// TIA Portal V17 export
// export: Created 2022-07-20T07:01:32.5794371Z, ExportSetting WithDefaults, DisplayName Totally Integrated Automation Portal, DisplayVersion V17, DisplayName TIA Portal Openness, DisplayVersion V17, DisplayName TIA Portal Version Control Interface, DisplayVersion V17, DisplayName SINAMICS Startdrive Advanced, DisplayVersion V17, DisplayName SINAMICS Startdrive G130, G150, S120, S150, SINAMICS MV, S210, DisplayVersion V17, DisplayName SINAMICS Startdrive G110M, G120, G120C, G120D, G120P, G115D, DisplayVersion V17, DisplayName STEP 7 Professional, DisplayVersion V17, DisplayName STEP 7 Safety, DisplayVersion V17, DisplayName WinCC Advanced, DisplayVersion V17
FUNCTION_BLOCK "FB10344_WebGuideProfinet"   // FB10344, LAD
TITLE = FB10342_WebGuide
{ S7_Optimized_Access := 'TRUE' }
VERSION : 0.1
// stored: AutoNumber false, IsIECCheckEnabled false, IsRetainMemResEnabled false, MemoryReserve 100, SetENOAutomatically false, UDAEnableTagReadback false
   VAR_INPUT
      RequestAcknowledge : Bool;
      Parameters : "stWebGuidePNParameters";
      CommInWebGuide_0 : Int;
      CommInWebGuide_1 : Int;
      CommInWebGuide_2 : Int;
      CommInWebGuide_3 : Int;
      CommInWebGuide_4 : Int;
      CommInWebGuide_5 : Int;
      CommInWebGuide_6 : Int;
      CommInWebGuide_7 : Int;
      CommInWebGuide_8 : Int;
      CommInWebGuide_9 : Int;
      CommInWebGuide_10 : Int;
      CommInWebGuide_11 : Int;
      CommInWebGuide_12 : Int;
      CommInWebGuide_13 : Int;
      CommInWebGuide_14 : Int;
      CommInWebGuide_15 : Int;
      CommInWebGuide_16 : Int;
      CommInWebGuide_17 : Int;
      CommInWebGuide_18 : Int;
      CommInWebGuide_19 : Int;
      CommInWebGuide_20 : Int;
      CommInWebGuide_21 : Int;
      CommInWebGuide_22 : Int;
      CommInWebGuide_23 : Int;
      CommInWebGuide_24 : Int;
      CommInWebGuide_25 : Int;
      CommInWebGuide_26 : Int;
      CommInWebGuide_27 : Int;
      CommInWebGuide_28 : Int;
   END_VAR
   VAR_OUTPUT
      CommOutWebGuide_0 : Int;
      CommOutWebGuide_1 : Int;
      CommOutWebGuide_2 : Int;
      CommOutWebGuide_3 : Int;
      CommOutWebGuide_4 : Int;
      CommOutWebGuide_5 : Int;
      CommOutWebGuide_6 : Int;
      CommOutWebGuide_7 : Int;
      CommOutWebGuide_8 : Int;
      CommOutWebGuide_9 : Int;
      CommOutWebGuide_10 : Int;
      CommOutWebGuide_11 : Int;
      CommOutWebGuide_12 : Int;
      CommOutWebGuide_13 : Int;
      CommOutWebGuide_14 : Int;
      CommOutWebGuide_15 : Int;
      CommOutWebGuide_16 : Int;
      CommOutWebGuide_17 : Int;
      CommOutWebGuide_18 : Int;
      CommOutWebGuide_19 : Int;
      CommOutWebGuide_20 : Int;
      CommOutWebGuide_21 : Int;
      CommOutWebGuide_22 : Int;
      CommOutWebGuide_23 : Int;
      CommOutWebGuide_24 : Int;
      CommOutWebGuide_25 : Int;
      CommOutWebGuide_26 : Int;
      CommOutWebGuide_27 : Int;
      CommOutWebGuide_28 : Int;
   END_VAR
   VAR_IN_OUT
      Requests : "stWebGuidePNRequests";
      States : "stWebGuidePNStates";
   END_VAR
   VAR
      RequestInternTrigger : Bool;
      R_Trig_Trigger : R_TRIG;
   END_VAR
BEGIN

REGION Network 1 (SCL): First Scan
   IF "FirstScan" THEN
       ;
   END_IF;
END_REGION

REGION Network 2 (SCL): Edge Signals & Timers
   REGION EDGE SIGNALS
       #R_Trig_Trigger(CLK := #RequestInternTrigger);

   END_REGION

   REGION TIMERS

   END_REGION
END_REGION

REGION Network 3 (SCL): Toogle
   IF #CommInWebGuide_0 < 16#7FFF THEN
       #CommOutWebGuide_0 := #CommInWebGuide_0 + 1;
   ELSE
       #CommOutWebGuide_0 := 0;
   END_IF;
END_REGION

REGION Network 4 (SCL): Web Speed [dm/min]
   #CommOutWebGuide_1 := #Parameters.WebSpeed;
   #States.WebSpeed := #CommInWebGuide_1;
   #States.LeftSensorPositionRead := #CommInWebGuide_14;
END_REGION

REGION Network 5 (SCL): WebGuide Mode

   IF #Requests.AutoMode AND NOT #States.AutomaticModeSelected THEN

       #CommOutWebGuide_2.%X0 := 1;
       #CommOutWebGuide_2.%X1 := 0;
       #CommOutWebGuide_2.%X2 := 0;
       #CommOutWebGuide_2.%X3 := TRUE;

   ELSIF #Requests.CenterMode AND NOT #States.CenterModeSelected THEN

       #CommOutWebGuide_2.%X0 := 0;
       #CommOutWebGuide_2.%X1 := 1;
       #CommOutWebGuide_2.%X2 := 0;
       #CommOutWebGuide_2.%X3 := TRUE;

   ELSIF #Requests.ManualMode AND NOT #States.ManualModeSelected THEN

       #CommOutWebGuide_2.%X0 := 0;
       #CommOutWebGuide_2.%X1 := 0;
       #CommOutWebGuide_2.%X2 := 1;
       #CommOutWebGuide_2.%X3 := TRUE;
   ELSE

       #CommOutWebGuide_2.%X0 := 0;
       #CommOutWebGuide_2.%X1 := 0;
       #CommOutWebGuide_2.%X2 := 0;
       #CommOutWebGuide_2.%X3 := 0;

   END_IF;

   #States.AutomaticModeSelected := #CommInWebGuide_2.%X0;
   #States.CenterModeSelected := #CommInWebGuide_2.%X1;
   #States.ManualModeSelected := #CommInWebGuide_2.%X2;
END_REGION

REGION Network 6 (SCL): WebGuide Web Offset

   IF #Requests.SetWebOffset AND #States.WebOffset<> #Parameters.WebOffset THEN

       #CommOutWebGuide_6 := #Parameters.WebOffset;
       #CommOutWebGuide_4.%X0 := TRUE;
   ELSE

       #CommOutWebGuide_4.%X0 := FALSE;

   END_IF;

   #States.WebOffset := #CommInWebGuide_11;
END_REGION

REGION Network 7 (SCL): WebGuide Target Position

   IF #Requests.SetTargetPosition THEN

       #CommOutWebGuide_7 := #Parameters.TargetPosition;
       #CommOutWebGuide_4.%X1 := TRUE;
   ELSE

       #CommOutWebGuide_4.%X1 := FALSE;

   END_IF;

   #States.ActualPosition := #CommInWebGuide_10;
   #States.CurrentGuidingPosition := #CommInWebGuide_12;
END_REGION

REGION Network 8 (SCL): WebGuide Set Center Position

   IF #Requests.SetCenterPosition THEN

       #CommOutWebGuide_10 := #Parameters.CenterPosition;
       #CommOutWebGuide_4.%X4 := TRUE;
   ELSE

       #CommOutWebGuide_4.%X4 := FALSE;

   END_IF;
   #States.WebCenterPosition := #CommInWebGuide_9;
END_REGION

REGION Network 9 (SCL): WebGuide Oscillations

   IF #Requests.ActivationOscillation THEN
       #CommOutWebGuide_4.%X5 := TRUE;
   ELSE
       #CommOutWebGuide_4.%X5 := FALSE;
   END_IF;

   IF #Requests.ChangeOscillationParameters THEN
       #CommOutWebGuide_20 := #Parameters.OscillationAmplitude;
       #CommOutWebGuide_21 := #Parameters.OscillationTime;
       #CommOutWebGuide_22 := #Parameters.OscillationWaveForm;

       #CommOutWebGuide_4.%X6 := TRUE;
   ELSE
       #CommOutWebGuide_4.%X6 := FALSE;
   END_IF;


   #States.OscillationModeActive := #CommInWebGuide_4.%X5;
END_REGION

REGION Network 10 (SCL): States
END_REGION
END_FUNCTION_BLOCK
